RoboDK station: AROB_AS6_A2_Testat.rdk

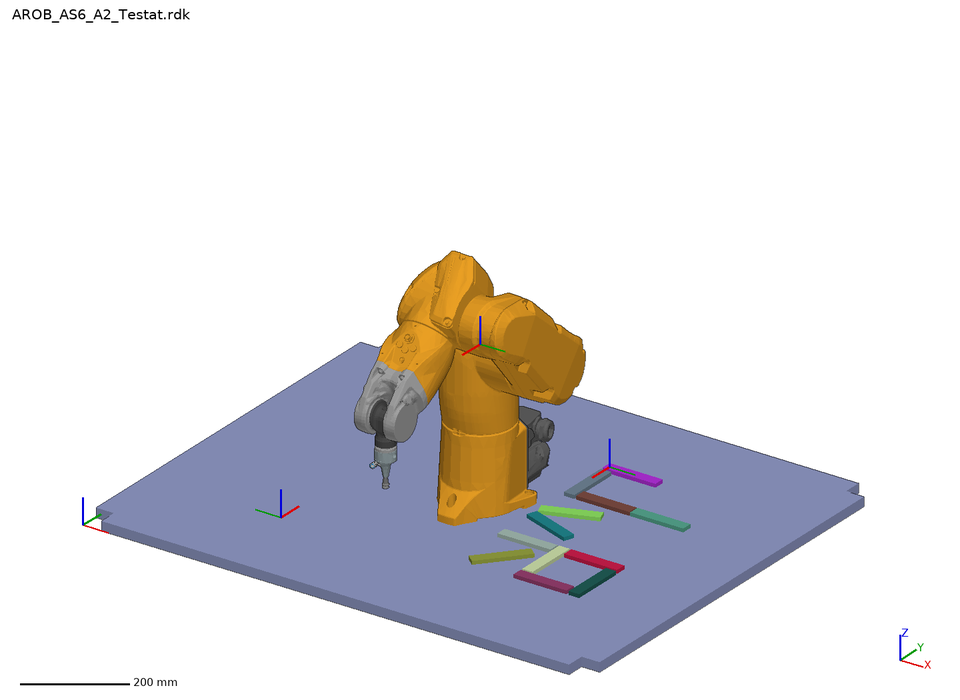
[picture v0: the station drawn from its stored meshes, robots at their saved joint values, targets as dots, program paths as lines]
Station AROB_AS6_A2_Testat (saved by RoboDK 5.6.9). Poses are relative to the parent item; angles as X-Y-Z fixed-axis rotations.
  - frame world at (0, 0, 0) mm
    - frame Staubli TX2-40 Base at (560, 460, 340) mm, rotated rx 0 ry 0 rz -90 deg
      - robot Staubli TX2-40: 6 axes, payload 1.7 kg, reach 515 mm, repeatability 0.02 mm, weight 29 kg
          modified DH rows (alpha deg, a mm, theta deg, d mm): 0, 0, 0, 320; -90, 0, -90, 35; 0, 225, -90, 0; -90, 0, 0, 225; 90, 0, 0, 0; -90, 0, 180, 65
          base shift (0, 0, -320) mm
          joint limits [-180, -125, -138, -270, -120, -270] to [180, 125, 138, 270, 133.5, 270]; home [0, 0, 90, 0, 0, 0]; saved at [0, 50.601, 77.88, 0, 51.518, 0]
        - tool LWS_VakuumGreifer_11, TCP at (0, 0, 77.8) mm, size 81.8 x 42 x 49.7 mm, geometry from LWS_VakuumGreifer_11.stp
    - frame pick at (300, 200, 20) mm, rotated rx 0 ry 0 rz 90 deg
    - frame place at (670, 715, 20) mm, rotated rx 0 ry 0 rz -90 deg
      - object block1 at (134.55, 206.55, 0) mm, rotated rx 180 ry 0 rz -90 deg, size 117.7 x 23.1 x 7.8 mm, geometry from block.stl
      - object block2 at (134.55, 86.55, 0) mm, rotated rx 180 ry 0 rz -90 deg, size 117.7 x 23.1 x 7.8 mm, geometry from block.stl
      - object block3 at (87.2, 11.55, 0) mm, rotated rx 180 ry 0 rz 180 deg, size 117.7 x 23.1 x 7.8 mm, geometry from block.stl
      - object block4 at (11.55, 58.55, 0) mm, rotated rx -180 ry 0 rz -90 deg, size 117.7 x 23.1 x 7.8 mm, geometry from block.stl
      - object block5 at (204.55, 56.55, 0) mm, rotated rx -180 ry 0 rz -70 deg, size 117.7 x 23.1 x 7.8 mm, geometry from block.stl
      - object block6 at (269.55, 56.55, 0) mm, rotated rx 180 ry 0 rz -110 deg, size 117.7 x 23.1 x 7.8 mm, geometry from block.stl
      - object block7 at (344.55, 58.55, 0) mm, rotated rx -180 ry 0 rz -90 deg, size 117.7 x 23.1 x 7.8 mm, geometry from block.stl
      - object block8 at (344.55, 206.55, 0) mm, rotated rx -180 ry 0 rz -90 deg, size 117.7 x 23.1 x 7.8 mm, geometry from block.stl
      - object block9 at (419.55, 255, 0) mm, rotated rx -180 ry 0 rz 180 deg, size 117.7 x 23.1 x 7.8 mm, geometry from block.stl
      - object block10 at (467.05, 179.95, 0) mm, rotated rx 180 ry 0 rz 90 deg, size 117.7 x 23.1 x 7.8 mm, geometry from block.stl
      - object block11 at (392.05, 132.55, 0) mm, rotated rx 180 ry 0 rz -180 deg, size 117.7 x 23.1 x 7.8 mm, geometry from block.stl
      - object block12 at (424.55, 56.55, 0) mm, rotated rx 180 ry 0 rz -40 deg, size 117.7 x 23.1 x 7.8 mm, geometry from block.stl
    - object reference_block at (0, 0, 0) mm, rotated rx 180 ry 0 rz 180 deg, size 117.7 x 23.1 x 7.8 mm, geometry from block.stl
    - object Arbeitsflaeche_geteilt at (0, 0, 0) mm, size 1120 x 920 x 20 mm, geometry from Arbeitsflaeche_geteilt.iges
    - object Arbeitsflaeche_komplett at (0, 0, 0) mm, size 1120 x 920 x 20 mm, geometry from Arbeitsflaeche_komplett.IGS
    - object Zelle at (0, 0, 0) mm, rotated rx 90 ry 0 rz -90 deg, size 1120 x 1947.8 x 1200 mm, geometry from Zelle.stp
  - Python program AddBlocks (listed below)
  - Python program DeleteBlocks (listed below)
  - Python program WriteLetters (listed below)

--- Python program AddBlocks ---
# Type help("robodk.robolink") or help("robodk.robomath") for more information
# Press F5 to run the script
# Documentation: https://robodk.com/doc/en/RoboDK-API.html
# Reference:     https://robodk.com/doc/en/PythonAPI/robodk.html
# Note: It is not required to keep a copy of this file, your Python script is saved with your RDK project

# You can also use the new version of the API:
import robodk.robolink as rl    # RoboDK API
import robodk.robomath as rm    # Robot toolbox
import numpy as np

RDK = rl.Robolink()

KAPLA_HEIGHT : int = 7.75
KAPLA_LENGTH : int = 117.70
KAPLA_WIDTH : int = 23.10

SPACING_TCP_BLOCK_HOVER = 30 # [mm] : Spacing between the TCP & Block.
SPACING_X_BLOCKS = 25 # [mm] : Spacing between the blocks.
SPACING_Y_BLOCKS = 120 # [mm] : Spacing between the blocks.

robot = RDK.Item('Staubli TX2-40', rl.ITEM_TYPE_ROBOT)
tool = RDK.Item('LWS_VakuumGreifer_11', rl.ITEM_TYPE_TOOL)
world = RDK.Item('world', rl.ITEM_TYPE_FRAME)
pick = RDK.Item('pick', rl.ITEM_TYPE_FRAME)
place = RDK.Item('place', rl.ITEM_TYPE_FRAME)

reference_block = RDK.Item('reference_block', rl.ITEM_TYPE_OBJECT)
n_blocks : int = 12
blocks = [None] * n_blocks

# [Prepare Pick Frame]
# Copy reference block...
reference_block.Copy()

rng = np.random.default_rng()
for i in range(0,n_blocks):
    # ...paste the blocks, rename it...
    blocks[i] = RDK.Paste().setName('block'+str(i + 1))
    # ..., set its reference frame...
    blocks[i].setParentStatic(pick)
    blocks[i].setColor([rng.random(), rng.random(), rng.random()])
    # ..., set its position (+ correct orientation)...
    blocks[i].setPose(rm.Staubli_2_Pose([SPACING_X_BLOCKS * i,0,0,0,180,90]))
    # ...and set its visibility
    blocks[i].setVisible(visible=True, visible_frame=False)

--- Python program DeleteBlocks ---
# Type help("robodk.robolink") or help("robodk.robomath") for more information
# Press F5 to run the script
# Documentation: https://robodk.com/doc/en/RoboDK-API.html
# Reference:     https://robodk.com/doc/en/PythonAPI/robodk.html
# Note: It is not required to keep a copy of this file, your Python script is saved with your RDK project

# You can also use the new version of the API:
import robodk.robolink as rl    # RoboDK API
import robodk.robomath as rm    # Robot toolbox
import numpy as np

RDK = rl.Robolink()

KAPLA_HEIGHT : int = 7.75
KAPLA_LENGTH : int = 117.70
KAPLA_WIDTH : int = 23.10

SPACING_TCP_BLOCK_HOVER = 30 # [mm] : Spacing between the TCP & Block.
SPACING_WIDTH_BLOCKS = 25 # [mm] : Spacing between the blocks.

robot = RDK.Item('Staubli TX2-40')
world = RDK.Item('world', rl.ITEM_TYPE_FRAME)
pick = RDK.Item('pick', rl.ITEM_TYPE_FRAME)
place = RDK.Item('place', rl.ITEM_TYPE_FRAME)

target_list_names = RDK.ItemList(filter=rl.ITEM_TYPE_OBJECT,list_names=True)

for target_name in target_list_names:
    if 'block' in target_name and target_name != 'reference_block':
        RDK.Delete(RDK.Item(target_name))

--- Python program WriteLetters ---
# Type help("robodk.robolink") or help("robodk.robomath") for more information
# Press F5 to run the script
# Documentation: https://robodk.com/doc/en/RoboDK-API.html
# Reference:     https://robodk.com/doc/en/PythonAPI/robodk.html
# Note: It is not required to keep a copy of this file, your Python script is saved with your RDK project

# You can also use the new version of the API:
import robodk.robolink as rl    # RoboDK API
import robodk.robomath as rm    # Robot toolbox
import numpy as np

RDK = rl.Robolink()

KAPLA_HEIGHT : int = 7.8
KAPLA_LENGTH : int = 117.70
KAPLA_WIDTH : int = 23.10

SPACING_TCP_BLOCK_HOVER = 30 # [mm] : Spacing between the TCP & Block.
SPACING_X_BLOCKS = 25 # [mm] : Spacing between the blocks.
SPACING_Y_BLOCKS = 120 # [mm] : Spacing between the blocks.



letter_block_positions = [
    # Letter J
    rm.Staubli_2_Pose([ 134.550, 206.550, KAPLA_HEIGHT, 180.000, 0.000,   0.000]), # Part 1: J  1
    rm.Staubli_2_Pose([ 134.550,  86.550, KAPLA_HEIGHT, 180.000, 0.000,   0.000]), # Part 2: J  2
    rm.Staubli_2_Pose([  87.200,  11.550, KAPLA_HEIGHT, 180.000, 0.000,  90.000]), # Part 3: J  3
    rm.Staubli_2_Pose([  11.550,  58.550, KAPLA_HEIGHT, 180.000, 0.000,   0.000]), # Part 4: J  4
    # Letter v
    rm.Staubli_2_Pose([ 204.550,  56.550, KAPLA_HEIGHT, 180.000, 0.000, -20.000]), # Part 1: v  5
    rm.Staubli_2_Pose([ 269.550,  56.550, KAPLA_HEIGHT, 180.000, 0.000,  20.000]), # Part 2: v  6
    # Letter R
    rm.Staubli_2_Pose([ 344.550,  58.550, KAPLA_HEIGHT, 180.000, 0.000,   0.000]), # Part 1: R  7
    rm.Staubli_2_Pose([ 344.550, 206.550, KAPLA_HEIGHT, 180.000, 0.000,   0.000]), # Part 2: R  8
    rm.Staubli_2_Pose([ 419.550, 255.000, KAPLA_HEIGHT, 180.000, 0.000,  90.000]), # Part 4: R  9
    rm.Staubli_2_Pose([ 467.050, 179.950, KAPLA_HEIGHT, 180.000, 0.000, 180.000]), # Part 6: R 10
    rm.Staubli_2_Pose([ 392.050, 132.550, KAPLA_HEIGHT, 180.000, 0.000,  90.000]), # Part 7: R 11
    rm.Staubli_2_Pose([ 424.550,  56.550, KAPLA_HEIGHT, 180.000, 0.000, -50.000]), # Part 8: R 12
]


robot = RDK.Item('Staubli TX2-40', rl.ITEM_TYPE_ROBOT)
tool = RDK.Item('LWS_VakuumGreifer_11', rl.ITEM_TYPE_TOOL)
world = RDK.Item('world', rl.ITEM_TYPE_FRAME)
pick = RDK.Item('pick', rl.ITEM_TYPE_FRAME)
place = RDK.Item('place', rl.ITEM_TYPE_FRAME)

midpoint = rm.Staubli_2_Pose([   595.000000,   110.000000,   200.000000,   -180.000000,     0.000000,   -90.000000 ])
robot.setAccelerationJoints(10)
robot.setSpeedJoints(20)


# [PICK & PLACE]
# Important is the spacing between the blocks and the amount of blocks
SPACING_X_BLOCKS = 25 # [mm] : Spacing between the blocks.
n_blocks : int = 12


robot.setPoseFrame(world)
robot.MoveJ(midpoint)

for i in range(0,n_blocks):
    # [PICKING]
    # jump to pick frame
    robot.setPoseFrame(pick)
    # move robot over the respective block
    robot.MoveJ(rm.Staubli_2_Pose([SPACING_X_BLOCKS * i, 0.0, SPACING_TCP_BLOCK_HOVER, 180.000, 0, 180.000]))
    # move onto block
    robot.MoveL(rm.Staubli_2_Pose([SPACING_X_BLOCKS * i, 0.0, KAPLA_HEIGHT, 180.000, 0, 180.000]))
    # pick it up
    tool.AttachClosest()
    # move back up
    robot.MoveL(rm.Staubli_2_Pose([SPACING_X_BLOCKS * i, 0.0, SPACING_TCP_BLOCK_HOVER, 180.000, 0, 180.000]))
    # move to the mid point / transfer point
    robot.setPoseFrame(world)
    robot.MoveJ(midpoint)

    # [PLACING]
    # jump to place frame
    robot.setPoseFrame(place)
    # move robot over the respective block
    robot.MoveJ(letter_block_positions[i] * rm.transl(0,0,-SPACING_TCP_BLOCK_HOVER))
    # move onto block
    robot.MoveJ(letter_block_positions[i])
    # place it by detaching
    tool.DetachAll(parent=place)
    # move robot back up
    robot.MoveJ(letter_block_positions[i] * rm.transl(0,0,-SPACING_TCP_BLOCK_HOVER))
    # move to the mid point / transfer point
    robot.setPoseFrame(world)
    robot.MoveJ(midpoint)

    # rinse and repeat
